{attribute 'qualified_only'}
{attribute 'strict'}
TYPE AxisParameters :
(
(* PLCopen specific parameters *) (* Index-Group 0x4000 + ID*)
    CommandedPosition       := 1,    (* lreal *) (* taken from NcToPlc *)
    SWLimitPos              := 2,    (* lreal *) (* IndexOffset= 16#0001_000E *)
    SWLimitNeg              := 3,    (* lreal *) (* IndexOffset= 16#0001_000D *)
    EnableLimitPos          := 4,    (* bool  *) (* IndexOffset= 16#0001_000C *)
    EnableLimitNeg          := 5,    (* bool  *) (* IndexOffset= 16#0001_000B *)
    EnablePosLagMonitoring  := 6,    (* bool  *) (* IndexOffset= 16#0002_0010 *)
    MaxPositionLag          := 7,    (* lreal *) (* IndexOffset= 16#0002_0012 *)
    MaxVelocitySystem       := 8,    (* lreal *) (* IndexOffset= 16#0000_0027 *)
    MaxVelocityAppl         := 9,    (* lreal *) (* IndexOffset= 16#0000_0027 *)
    ActualVelocity          := 10,   (* lreal *) (* taken from NcToPlc *)
    CommandedVelocity       := 11,   (* lreal *) (* taken from NcToPlc *)
    MaxAccelerationSystem   := 12,   (* lreal *) (* IndexOffset= 16#0000_0101 *)
    MaxAccelerationAppl     := 13,   (* lreal *) (* IndexOffset= 16#0000_0101 *)
    MaxDecelerationSystem   := 14,   (* lreal *) (* IndexOffset= 16#0000_0102 *)
    MaxDecelerationAppl     := 15,   (* lreal *) (* IndexOffset= 16#0000_0102 *)
    MaxJerkSystem           := 16,   (* lreal *) (* IndexOffset= 16#0000_0103 *)
    MaxJerkAppl             := 17,   (* lreal *) (* IndexOffset= 16#0000_0103 *)

(* Beckhoff specific parameters *) (* Index-Group 0x4000 + ID*)
   AxisId := 1000,                   (* lreal *) (* IndexOffset= 16#0000_0001 *)
   AxisVeloManSlow,                  (* lreal *) (* IndexOffset= 16#0000_0008 *)
   AxisVeloManFast,                  (* lreal *) (* IndexOffset= 16#0000_0009 *)
   AxisVeloMax,                      (* lreal *) (* IndexOffset= 16#0000_0027 *)
   AxisAcc,                          (* lreal *) (* IndexOffset= 16#0000_0101 *)
   AxisDec,                          (* lreal *) (* IndexOffset= 16#0000_0102 *)
   AxisJerk,                         (* lreal *) (* IndexOffset= 16#0000_0103 *)
   MaxJerk,                          (* lreal *) (* IndexOffset= 16#0000_0103 *)
   AxisMaxVelocity,                  (* lreal *) (* IndexOffset= 16#0000_0027 *)
   AxisRapidTraverseVelocity,        (* lreal *) (* IndexOffset= 16#0000_000A *)
   AxisManualVelocityFast,           (* lreal *) (* IndexOffset= 16#0000_0009 *)
   AxisManualVelocitySlow,           (* lreal *) (* IndexOffset= 16#0000_0008 *)
   AxisCalibrationVelocityForward,   (* lreal *) (* IndexOffset= 16#0000_0006 *)
   AxisCalibrationVelocityBackward,  (* lreal *) (* IndexOffset= 16#0000_0007 *)
   AxisJogIncrementForward,          (* lreal *) (* IndexOffset= 16#0000_0018 *)
   AxisJogIncrementBackward,         (* lreal *) (* IndexOffset= 16#0000_0019 *)
   AxisEnMinSoftPosLimit,            (* bool  *) (* IndexOffset= 16#0001_000B *)
   AxisMinSoftPosLimit,              (* lreal *) (* IndexOffset= 16#0001_000D *)
   AxisEnMaxSoftPosLimit,            (* bool  *) (* IndexOffset= 16#0001_000C *)
   AxisMaxSoftPosLimit,              (* lreal *) (* IndexOffset= 16#0001_000E *)
   AxisEnPositionLagMonitoring,      (* bool  *) (* IndexOffset= 16#0002_0010 *)
   AxisMaxPosLagValue,               (* lreal *) (* IndexOffset= 16#0002_0012 *)
   AxisMaxPosLagFilterTime,          (* lreal *) (* IndexOffset= 16#0002_0013 *)
   AxisEnPositionRangeMonitoring,    (* bool  *) (* IndexOffset= 16#0000_000F *)
   AxisPositionRangeWindow,          (* lreal *) (* IndexOffset= 16#0000_0010 *)
   AxisEnTargetPositionMonitoring,   (* bool  *) (* IndexOffset= 16#0000_0015 *)
   AxisTargetPositionWindow,         (* lreal *) (* IndexOffset= 16#0000_0016 *)
   AxisTargetPositionMonitoringTime, (* lreal *) (* IndexOffset= 16#0000_0017 *)
   AxisEnInTargetTimeout,            (* bool  *) (* IndexOffset= 16#0000_0029 *)
   AxisInTargetTimeout,              (* lreal *) (* IndexOffset= 16#0000_002A *)
   AxisEnMotionMonitoring,           (* bool  *) (* IndexOffset= 16#0000_0011 *)
   AxisMotionMonitoringWindow,       (* lreal *) (* IndexOffset= 16#0000_0028 *)
   AxisMotionMonitoringTime,         (* lreal *) (* IndexOffset= 16#0000_0012 *)
   AxisDelayTimeVeloPosition,        (* lreal *) (* IndexOffset= 16#0000_0104 *)
   AxisEnLoopingDistance,            (* bool  *) (* IndexOffset= 16#0000_0013 *)
   AxisLoopingDistance,              (* lreal *) (* IndexOffset= 16#0000_0014 *)
   AxisEnBacklashCompensation,       (* bool  *) (* IndexOffset= 16#0000_002B *)
   AxisBacklash,                     (* lreal *) (* IndexOffset= 16#0000_002C *)
   AxisEnDataPersistence,            (* bool  *) (* IndexOffset= 16#0000_0030 *)
   AxisRefVeloOnRefOutput,           (* lreal *) (* IndexOffset= 16#0003_0101 *)
   AxisOverrideType,                 (* lreal *) (* IndexOffset= 16#0000_0105 *)
   (* new since 4/2007 *)
   AxisEncoderScalingFactor,         (* lreal *) (* IndexOffset= 16#0001_0006 *)
   AxisEncoderOffset,                (* lreal *) (* IndexOffset= 16#0001_0007 *)
   AxisEncoderDirectionInverse,      (* bool  *) (* IndexOffset= 16#0001_0008 *)
   AxisEncoderMask,                  (* dword *) (* IndexOffset= 16#0001_0015 *)
   AxisEncoderModuloValue,           (* lreal *) (* IndexOffset= 16#0001_0009 *)
   AxisModuloToleranceWindow,        (* lreal *) (* IndexOffset= 16#0001_001B *)
   AxisEnablePosCorrection,          (* bool  *) (* IndexOffset= 16#0001_0016 *)
   AxisPosCorrectionFilterTime,      (* lreal *) (* IndexOffset= 16#0001_0017 *)
   (* new since 1/2010 *)
   AxisUnitInterpretation,           (* lreal *) (* IndexOffset= 16#0000_0026 *)
   AxisMotorDirectionInverse,        (* bool  *) (* IndexOffset= 16#0003_0006 *)
   (* new since 1/2011 *)
   AxisCycleTime,                    (* lreal *) (* IndexOffset= 16#0000_0004 *)
   (* new since 5/2011 *)
   AxisFastStopSignalType,           (* dword *) (* IndexOffset= 16#0000_001E *)
   AxisFastAcc,                      (* lreal *) (* IndexOffset= 16#0000_010A *)
   AxisFastDec,                      (* lreal *) (* IndexOffset= 16#0000_010B *)
   AxisFastJerk,                     (* lreal *) (* IndexOffset= 16#0000_010C *)

(* Beckhoff specific axis status information - READ ONLY *) (* Index-Group 0x4100 + ID*)
   AxisTargetPosition := 2000,       (* lreal *) (* IndexOffset= 16#0000_0013 *)
   AxisRemainingTimeToGo,            (* lreal *) (* IndexOffset= 16#0000_0014 *)
   AxisRemainingDistanceToGo,        (* lreal *) (* IndexOffset= 16#0000_0022, 16#0000_0042 *)

(* Beckhoff specific axis functions *)
   (* read/write gear ratio of a slave *)
   AxisGearRatio := 3000,            (* lreal *) (* read: IndexGroup=0x4100+ID, IdxOffset=16#0000_0022, *)
                   (* write:IndexGroup=0x4200+ID, IdxOffset=16#0000_0042 *)

(* Beckhoff specific other parameters *)
   (* new since 1/2011 *)
   NcSafCycleTime := 4000,           (* lreal *) (* IndexOffset= 16#0000_0010 *)
   NcSvbCycleTime                    (* lreal *) (* IndexOffset= 16#0000_0012 *)

);
END_TYPE

(* stored: Version 1.1.0.1, ProductVersion 3.1.4024.0
   EnumerationTextList AxisParameters: Id {9199cc42-106a-4663-aaa5-d49855d9aa9f} *)
